# EPICS autosave request: iocBoot/iocddrive/auto_positions.req
file motor_positions.req P=MLL:ddrive:,M=m1
